SYSTEM TEST_CSW (* Test CLIENTW/SERVERW Configuration *)
  (* Standard: 61499-1 *)
  (* Version 0.0, 2004-10-19, JHC, Rockwell Automation *)
  DEVICE CLIENT : FRAME_DEVICE
    RESOURCE RES1 : PANEL_RESOURCE
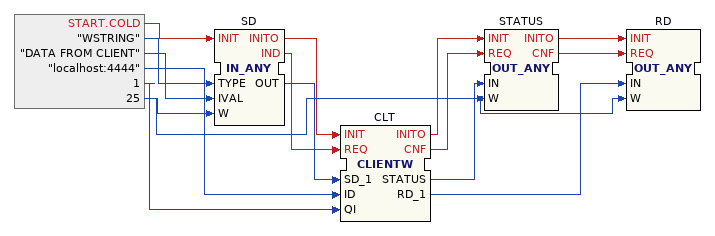
      FBS
        SD : IN_ANY;
        CLT : CLIENTW;
        STATUS : OUT_ANY;
        RD : OUT_ANY;
      END_FBS
      EVENT_CONNECTIONS
        START.COLD TO SD.INIT;
        SD.INITO TO CLT.INIT;
        SD.IND TO CLT.REQ;
        CLT.INITO TO STATUS.INIT;
        CLT.CNF TO STATUS.REQ;
        STATUS.INITO TO RD.INIT;
        STATUS.CNF TO RD.REQ;
      END_CONNECTIONS
      DATA_CONNECTIONS
        "WSTRING" TO SD.TYPE;
        "DATA FROM CLIENT" TO SD.IVAL;
        SD.OUT TO CLT.SD_1;
        "localhost:4444" TO CLT.ID;
        CLT.STATUS TO STATUS.IN;
        CLT.RD_1 TO RD.IN;
        1 TO CLT.QI;
        25 TO SD.W;
        25 TO STATUS.W;
        25 TO RD.W;
      END_CONNECTIONS
    END_RESOURCE
    DATA_CONNECTIONS
      3 TO RES1.ROWS;
      1 TO RES1.COLS;
    END_CONNECTIONS
  END_DEVICE
  DEVICE SERVER : FRAME_DEVICE
    RESOURCE RES1 : PANEL_RESOURCE
      FBS
        SD : IN_ANY;
        CLT : SERVERW;
        STATUS : OUT_ANY;
        RD : OUT_ANY;
        CONC : FB_CONCAT; (* Force WSTRING output to replace CLT.SD *)
      END_FBS
      EVENT_CONNECTIONS
        START.COLD TO SD.INIT;
        SD.INITO TO CLT.INIT;
        CLT.INITO TO STATUS.INIT;
        STATUS.INITO TO RD.INIT;
        STATUS.CNF TO RD.REQ;
        CLT.IND TO STATUS.REQ;
        SD.IND TO CONC.REQ;
        CONC.CNF TO CLT.RSP;
      END_CONNECTIONS
      DATA_CONNECTIONS
        "WSTRING" TO SD.TYPE;
        "DATA" TO SD.IVAL;
        CLT.STATUS TO STATUS.IN;
        CLT.RD_1 TO RD.IN;
        1 TO CLT.QI;
        25 TO SD.W;
        25 TO STATUS.W;
        25 TO RD.W;
        " FROM SERVER" TO CONC.IN2;
        SD.OUT TO CONC.IN1;
        CONC.OUT TO CLT.SD_1;
        "localhost:4444" TO CLT.ID;
      END_CONNECTIONS
    END_RESOURCE
    DATA_CONNECTIONS
      3 TO RES1.ROWS;
      1 TO RES1.COLS;
    END_CONNECTIONS
  END_DEVICE
  DATA_CONNECTIONS (* parameter values *)
    [100,100,150,125] TO CLIENT.BOUNDS;
    [250,100,150,125] TO SERVER.BOUNDS;
  END_CONNECTIONS
END_SYSTEM
